// TIA Portal V19 export
FUNCTION "SCALING" : Void   // FC3, LAD
{ S7_Optimized_Access := 'TRUE' }
// stored: SetENOAutomatically false
BEGIN

REGION Network 1: LT-1
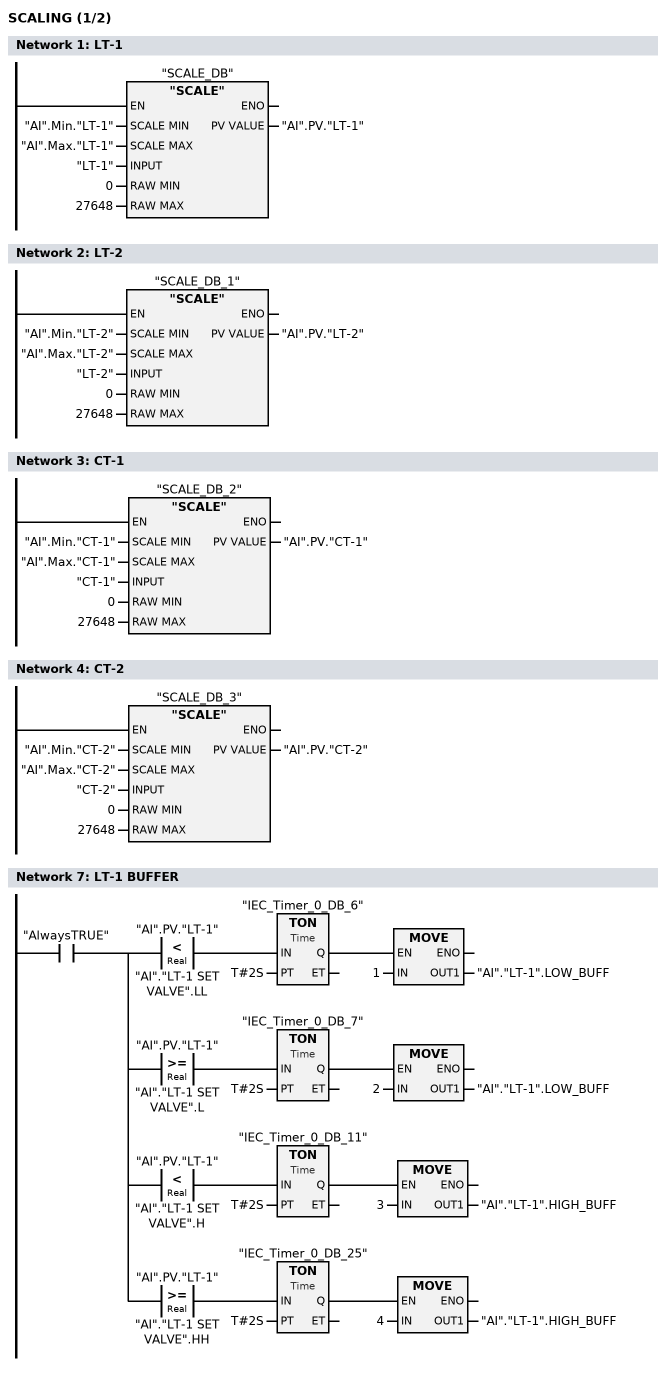
   RUNG wire#powerrail
      "SCALE_DB"("SCALE MIN" := "AI".Min."LT-1", "SCALE MAX" := "AI".Max."LT-1", INPUT := "LT-1", "RAW MIN" := 0, "RAW MAX" := 27648, "PV VALUE" => "AI".PV."LT-1")
   END_RUNG
   // the same network as SCL:
   "SCALE_DB"("SCALE MIN" := "AI".Min."LT-1",   // "SCALE"
              "SCALE MAX" := "AI".Max."LT-1",
              INPUT := "LT-1",
              "RAW MIN" := 0,
              "RAW MAX" := 27648,
              "PV VALUE" => "AI".PV."LT-1");
END_REGION

REGION Network 2: LT-2
   RUNG wire#powerrail
      "SCALE_DB_1"("SCALE MIN" := "AI".Min."LT-2", "SCALE MAX" := "AI".Max."LT-2", INPUT := "LT-2", "RAW MIN" := 0, "RAW MAX" := 27648, "PV VALUE" => "AI".PV."LT-2")
   END_RUNG
   // the same network as SCL:
   "SCALE_DB_1"("SCALE MIN" := "AI".Min."LT-2",   // "SCALE"
                "SCALE MAX" := "AI".Max."LT-2",
                INPUT := "LT-2",
                "RAW MIN" := 0,
                "RAW MAX" := 27648,
                "PV VALUE" => "AI".PV."LT-2");
END_REGION

REGION Network 3: CT-1
   RUNG wire#powerrail
      "SCALE_DB_2"("SCALE MIN" := "AI".Min."CT-1", "SCALE MAX" := "AI".Max."CT-1", INPUT := "CT-1", "RAW MIN" := 0, "RAW MAX" := 27648, "PV VALUE" => "AI".PV."CT-1")
   END_RUNG
   // the same network as SCL:
   "SCALE_DB_2"("SCALE MIN" := "AI".Min."CT-1",   // "SCALE"
                "SCALE MAX" := "AI".Max."CT-1",
                INPUT := "CT-1",
                "RAW MIN" := 0,
                "RAW MAX" := 27648,
                "PV VALUE" => "AI".PV."CT-1");
END_REGION

REGION Network 4: CT-2
   RUNG wire#powerrail
      "SCALE_DB_3"("SCALE MIN" := "AI".Min."CT-2", "SCALE MAX" := "AI".Max."CT-2", INPUT := "CT-2", "RAW MIN" := 0, "RAW MAX" := 27648, "PV VALUE" => "AI".PV."CT-2")
   END_RUNG
   // the same network as SCL:
   "SCALE_DB_3"("SCALE MIN" := "AI".Min."CT-2",   // "SCALE"
                "SCALE MAX" := "AI".Max."CT-2",
                INPUT := "CT-2",
                "RAW MIN" := 0,
                "RAW MAX" := 27648,
                "PV VALUE" => "AI".PV."CT-2");
END_REGION

REGION Network 7: LT-1 BUFFER
   RUNG wire#powerrail
      Contact( "AlwaysTRUE" )
      wire#w1
      { S7_Templates := "SrcType := Real" } LT_Contact(in1 := "AI".PV."LT-1", in2 := "AI"."LT-1 SET VALVE".LL)
      { S7_Templates := "time_type := Time" } "IEC_Timer_0_DB_6".TON(pt := T#2S, et =>)
      Move(in := 1, out1 => "AI"."LT-1".LOW_BUFF)
   END_RUNG
   RUNG wire#w1
      { S7_Templates := "SrcType := Real" } GE_Contact(in1 := "AI".PV."LT-1", in2 := "AI"."LT-1 SET VALVE".L)
      { S7_Templates := "time_type := Time" } "IEC_Timer_0_DB_7".TON(pt := T#2S, et =>)
      Move(in := 2, out1 => "AI"."LT-1".LOW_BUFF)
   END_RUNG
   RUNG wire#w1
      { S7_Templates := "SrcType := Real" } LT_Contact(in1 := "AI".PV."LT-1", in2 := "AI"."LT-1 SET VALVE".H)
      { S7_Templates := "time_type := Time" } "IEC_Timer_0_DB_11".TON(pt := T#2S, et =>)
      Move(in := 3, out1 => "AI"."LT-1".HIGH_BUFF)
   END_RUNG
   RUNG wire#w1
      { S7_Templates := "SrcType := Real" } GE_Contact(in1 := "AI".PV."LT-1", in2 := "AI"."LT-1 SET VALVE".HH)
      { S7_Templates := "time_type := Time" } "IEC_Timer_0_DB_25".TON(pt := T#2S, et =>)
      Move(in := 4, out1 => "AI"."LT-1".HIGH_BUFF)
   END_RUNG
   // the same network as SCL:
   "IEC_Timer_0_DB_6".TON(IN := "AlwaysTRUE" AND ("AI".PV."LT-1" < "AI"."LT-1 SET VALVE".LL), PT := T#2S);
   IF "IEC_Timer_0_DB_6".Q THEN "AI"."LT-1".LOW_BUFF := 1; END_IF;
   "IEC_Timer_0_DB_7".TON(IN := "AlwaysTRUE" AND ("AI".PV."LT-1" >= "AI"."LT-1 SET VALVE".L), PT := T#2S);
   IF "IEC_Timer_0_DB_7".Q THEN "AI"."LT-1".LOW_BUFF := 2; END_IF;
   "IEC_Timer_0_DB_11".TON(IN := "AlwaysTRUE" AND ("AI".PV."LT-1" < "AI"."LT-1 SET VALVE".H), PT := T#2S);
   IF "IEC_Timer_0_DB_11".Q THEN "AI"."LT-1".HIGH_BUFF := 3; END_IF;
   "IEC_Timer_0_DB_25".TON(IN := "AlwaysTRUE" AND ("AI".PV."LT-1" >= "AI"."LT-1 SET VALVE".HH), PT := T#2S);
   IF "IEC_Timer_0_DB_25".Q THEN "AI"."LT-1".HIGH_BUFF := 4; END_IF;
END_REGION

REGION Network 8: LT-2 BUFFER
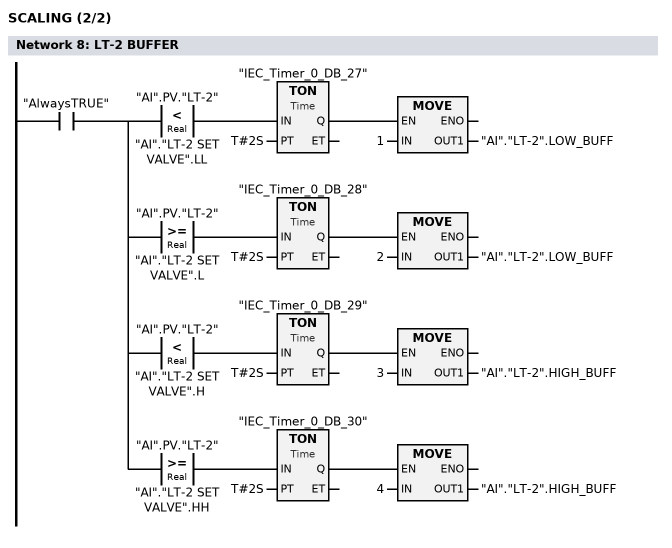
   RUNG wire#powerrail
      Contact( "AlwaysTRUE" )
      wire#w1
      { S7_Templates := "SrcType := Real" } LT_Contact(in1 := "AI".PV."LT-2", in2 := "AI"."LT-2 SET VALVE".LL)
      { S7_Templates := "time_type := Time" } "IEC_Timer_0_DB_27".TON(pt := T#2S, et =>)
      Move(in := 1, out1 => "AI"."LT-2".LOW_BUFF)
   END_RUNG
   RUNG wire#w1
      { S7_Templates := "SrcType := Real" } GE_Contact(in1 := "AI".PV."LT-2", in2 := "AI"."LT-2 SET VALVE".L)
      { S7_Templates := "time_type := Time" } "IEC_Timer_0_DB_28".TON(pt := T#2S, et =>)
      Move(in := 2, out1 => "AI"."LT-2".LOW_BUFF)
   END_RUNG
   RUNG wire#w1
      { S7_Templates := "SrcType := Real" } LT_Contact(in1 := "AI".PV."LT-2", in2 := "AI"."LT-2 SET VALVE".H)
      { S7_Templates := "time_type := Time" } "IEC_Timer_0_DB_29".TON(pt := T#2S, et =>)
      Move(in := 3, out1 => "AI"."LT-2".HIGH_BUFF)
   END_RUNG
   RUNG wire#w1
      { S7_Templates := "SrcType := Real" } GE_Contact(in1 := "AI".PV."LT-2", in2 := "AI"."LT-2 SET VALVE".HH)
      { S7_Templates := "time_type := Time" } "IEC_Timer_0_DB_30".TON(pt := T#2S, et =>)
      Move(in := 4, out1 => "AI"."LT-2".HIGH_BUFF)
   END_RUNG
   // the same network as SCL:
   "IEC_Timer_0_DB_27".TON(IN := "AlwaysTRUE" AND ("AI".PV."LT-2" < "AI"."LT-2 SET VALVE".LL), PT := T#2S);
   IF "IEC_Timer_0_DB_27".Q THEN "AI"."LT-2".LOW_BUFF := 1; END_IF;
   "IEC_Timer_0_DB_28".TON(IN := "AlwaysTRUE" AND ("AI".PV."LT-2" >= "AI"."LT-2 SET VALVE".L), PT := T#2S);
   IF "IEC_Timer_0_DB_28".Q THEN "AI"."LT-2".LOW_BUFF := 2; END_IF;
   "IEC_Timer_0_DB_29".TON(IN := "AlwaysTRUE" AND ("AI".PV."LT-2" < "AI"."LT-2 SET VALVE".H), PT := T#2S);
   IF "IEC_Timer_0_DB_29".Q THEN "AI"."LT-2".HIGH_BUFF := 3; END_IF;
   "IEC_Timer_0_DB_30".TON(IN := "AlwaysTRUE" AND ("AI".PV."LT-2" >= "AI"."LT-2 SET VALVE".HH), PT := T#2S);
   IF "IEC_Timer_0_DB_30".Q THEN "AI"."LT-2".HIGH_BUFF := 4; END_IF;
END_REGION
END_FUNCTION
